FUNCTION_BLOCK FB_AC
VAR_INPUT
	AC_IPAddr: STRING;
	ACcontrol: ST_ACcontrol;
END_VAR
VAR_OUTPUT
	ACstatus: ST_ACStatus;
END_VAR
VAR
	fbACcomm: FB_ACcomm;
	prevMode: INT;
	step: (eIdle, eOn, eOff, eModeChange, eError);
	fbOnCmd: FB_CommandHandling;
	fbOffCmd: FB_CommandHandling;
	fbModeChangeCmd: FB_CommandHandling;
END_VAR

VAR CONSTANT
	cOnCmd: STRING := 'AC On Cmd';
	cOffCmd: STRING := 'AC Off Cmd';
	cModeChangeCmd: STRING := 'AC Mode = ';
END_VAR


	fbACcomm( AC_IPAddr	:=	AC_IPAddr );
	
	fbOnCmd(cmd:= ACcontrol.OnCmd, timeoutOccured => , reset:= , timeout:= , Q=> );
	fbOffCmd(cmd:= ACcontrol.OffCmd, timeoutOccured => , reset:= , timeout:= , Q=> );
	fbModeChangeCmd(cmd:= ACcontrol.modeSelection <> prevMode, timeoutOccured => , reset:= , timeout:= , Q=> );
	prevMode	:=	ACcontrol.modeSelection;
	
	CASE step OF 
	eIdle: 
		IF fbOnCmd.Q THEN
			step		:=	eOn;
		END_IF
		IF fbOffCmd.Q THEN
			step		:=	eOff;
		END_IF
		IF fbModeChangeCmd.Q THEN
			step		:=	eModeChange;
		END_IF
			
	eOn:
		fbACcomm(sCmd:= cOnCmd, bSend:= TRUE);
		IF fbACcomm.bResponseReceived OR fbACcomm.bNoResponse THEN
			fbACcomm(sCmd:= , bSend:= FALSE );
			step		:=	eIdle;
		END_IF
		
	eOff:
		fbACcomm(sCmd:= cOffCmd, bSend:= TRUE);
		IF fbACcomm.bResponseReceived OR fbACcomm.bNoResponse THEN
			fbACcomm(sCmd:= , bSend:= FALSE );
			step		:=	eIdle;
		END_IF
		
	eModeChange:
		fbACcomm(sCmd:= CONCAT(cModeChangeCmd, INT_TO_STRING(ACcontrol.modeSelection)), bSend:= TRUE);
		IF fbACcomm.bResponseReceived OR fbACcomm.bNoResponse THEN
			fbACcomm(sCmd:= , bSend:= FALSE );
			step		:=	eIdle;
		END_IF
		
	eError:
	END_CASE
	
	
	
	
	
	
	(*
	IF ACcontrol.OnCmd THEN
		ACstatus.OnOff	:=	TRUE;
	END_IF
	IF ACcontrol.OffCmd THEN
		ACstatus.OnOff	:=	FALSE;
	END_IF
	
	ACstatus.mode	:= 	ACcontrol.modeSelection;	
	
	IF ACcontrol.swing.HorizOn THEN
		ACstatus.HorizSwingOnOff	:=	TRUE;
	END_IF
	IF ACcontrol.swing.HorizOff THEN
		ACstatus.HorizSwingOnOff	:=	FALSE;
	END_IF
	IF ACcontrol.swing.VertiOn THEN
		ACstatus.VertiSwingOnOff	:=	TRUE;
	END_IF
	IF ACcontrol.swing.VertiOff THEN
		ACstatus.VertiSwingOnOff	:=	FALSE;
	END_IF
	
	IF ACcontrol.tempUp THEN
		ACstatus.temp	:=	ACstatus.temp + 1;
	END_IF
	IF ACcontrol.tempDown THEN
		ACstatus.temp	:=	ACstatus.temp - 1;
	END_IF
	IF ACcontrol.tempSP <> ACcontrol.tempSP_prev THEN
		ACstatus.temp			:=	ACcontrol.tempSP;
		ACcontrol.tempSP_prev	:=	ACcontrol.tempSP;
	END_IF
	*)

END_FUNCTION_BLOCK

(* stored: Version 1.1.0.1, ProductVersion 3.1.4024.12
   POU FB_AC: Id {2dab7e2d-10a2-4e51-9a30-451f3dc56294}, SpecialFunc None *)
